(* IEC 61131-3 sources: volt/packages/volt-lsp-iec/test-corpus/lenze-mid/Device/Plc Logic/Application/Library Manager/L_FirstErrorCapture, 3.26.2.8 (Lenze), 36 files *)

(* ---- ENUMSTEPSFILEHANDLING.dut ---- *)
TYPE ENUMSTEPSFILEHANDLING :
(
	INIT := 0,
	OPENFILE := 1,
	GETSIZEFILE := 2,
	READFILE := 3,
	WAITREAD := 4,
	WAITCLOSE := 5,
	CLOSEFILE := 6,
	DONE := 7
);
END_TYPE

(* ---- SCCATEGORYSTRUCT.dut ---- *)
TYPE SCCATEGORYSTRUCT :
STRUCT
	ASSTR : ARRAY [0..uiNoOfDowntimeCategories] OF STRING(55);
	AXERROR : ARRAY [0..uiNoOfDowntimeCategories] OF BOOL;
END_STRUCT
END_TYPE

(* ---- SCERRORACCESS.dut ---- *)
TYPE SCERRORACCESS :
STRUCT
	DWCATEGORY : DWORD;
	WERRORCODE : WORD;
	ETYPE : INT;
	STEXT : STRING;
END_STRUCT
END_TYPE

(* ---- SCERRORDATA.dut ---- *)
TYPE SCERRORDATA :
STRUCT
	XFIRSTERRORACTIVE : BOOL;
	XISWARNINGINFO : BOOL;
	IPRIORITY : INT;
	DWERRORNUMBER : DWORD;
END_STRUCT
END_TYPE

(* ---- SCERRORDATA_BASE.dut ---- *)
TYPE SCERRORDATA_BASE :
STRUCT
	SERRDESC : STRING;
	SCATEGORYDESC : STRING(55);
	DWERRORCATEGORY : DWORD;
	IPRODUCTIONEVENTMODE : INT;
	XCATEGORYERROR : BOOL;
END_STRUCT
END_TYPE

(* ---- SCREADERRORFROMFILEIN.dut ---- *)
TYPE SCREADERRORFROMFILEIN :
STRUCT
	SFILENAME : FILE.CAA.FILENAME := 'SoftPlcParameter/SoftPlcParameter.lxd';
	IMAXREADLOOPS : INT := 1;
	WTEXTLISTID : WORD := 15360;
	WENDTEXTLISTID : WORD := 16383;
	WERRORID : WORD := 1;
END_STRUCT
END_TYPE

(* ---- SCREADERRORFROMFILEOUT.dut ---- *)
TYPE SCREADERRORFROMFILEOUT :
STRUCT
	WFINDTEXTLISTID : WORD;
	WFINDERRORID : WORD;
	DIREADROWS : DINT;
	DIERRORROWS : DINT;
	SERRORTEXT : STRING(255);
	XEOF : BOOL;
	TEXCUTETIME : TIME;
	STEP : enumStepsFileHandling;
	STATUS : scRearErrorfromFileStatus;
END_STRUCT
END_TYPE

(* ---- SCREARERRORFROMFILESTATUS.dut ---- *)
TYPE SCREARERRORFROMFILESTATUS :
STRUCT
	XDONEOPENFILE : BOOL;
	XBUSYOPENFILE : BOOL;
	XERROROPENFILE : BOOL;
	EOPENFILEERROR : FILE.ERROR;
	HFILE : FILE.CAA.HANDLE;
	XDONEGETSIZEFILE : BOOL;
	XBUSYGETSIZEFILE : BOOL;
	XERRORGETSIZEFILE : BOOL;
	EGETSIZEFILEERROR : FILE.ERROR;
	SZSIZE : FILE.CAA.SIZE;
	XDONEREADFILE : BOOL;
	XBUSYREADFILE : BOOL;
	XERRORREADFILE : BOOL;
	EREADFILEERROR : FILE.ERROR;
	XDONECLOSEFILE : BOOL;
	XBUSYCLOSEFILE : BOOL;
	XERRORCLOSEFILE : BOOL;
	ECLOSEFILEERROR : FILE.ERROR;
	XDONEFINDERROR : BOOL;
	XBUSYFINDERROR : BOOL;
	XERRORFINDERROR : BOOL;
END_STRUCT
END_TYPE

(* ---- SCTM_FB_ERROR.dut ---- *)
TYPE SCTM_FB_ERROR :
STRUCT
	XAXISERROR : BIT;
	XAXISWARNING : BIT;
	XDRIVEERROR : BIT;
	XDRIVEWARNING : BIT;
	IERRORID : INT;
	DWDRIVEERROR : DWORD;
END_STRUCT
END_TYPE

(* ---- UERRORNUMBER.dut ---- *)
TYPE UERRORNUMBER :
UNION
	DWERRORNUMBER : DWORD;
	AWERRORINFO : ARRAY [1..2] OF WORD;
END_UNION
END_TYPE

(* ---- GVL_ERRCAPT.gvl ---- *)
VAR_GLOBAL
	IUDINTQTY : INT := 4;
	IERRORQTY : INT := 160;
	IERRCATEGORY : INT := 99;
END_VAR

(* ---- GVL_FIRSTERRORLOCAL.gvl ---- *)
VAR_GLOBAL
	UINOOFDOWNTIMECATEGORIES : UINT := 99;
END_VAR

(* ---- GVL_READERRORFROMFILE.gvl ---- *)
VAR_GLOBAL
	IMAXERRORTEXTARRAYSIZE : INT := 1250;
	IMAXREADSIZE : INT := 80;
	ASERRORTEXT : ARRAY [0..GVL_ReadErrorFromFile.imaxErrorTextArraySize] OF STRING(255);
	ADWERRORID : ARRAY [0..GVL_ReadErrorFromFile.imaxErrorTextArraySize] OF DWORD;
END_VAR

(* ---- GETAPPLICATIONTERRORSTRING.pou ---- *)
FUNCTION GETAPPLICATIONTERRORSTRING : STRING(255)
VAR_INPUT
	WTEXTREFID : WORD;
	WERRORID : WORD;
	DWERRORNUMBER : DWORD;
END_VAR
END_FUNCTION

(* ---- GETDATETIMEFROMJSON.pou ---- *)
FUNCTION GETDATETIMEFROMJSON : STRING
VAR_INPUT
	XUSEMILLISECONDS : BOOL;
END_VAR
VAR_IN_OUT
	SJSONSTRING : STRING(255);
END_VAR
END_FUNCTION

(* ---- GETDRIVEERRORSTRING.pou ---- *)
FUNCTION GETDRIVEERRORSTRING : STRING(255)
VAR_INPUT
	WTEXTREFID : WORD;
	WERRORID : WORD;
	DWERRORNUMBER : DWORD;
END_VAR
END_FUNCTION

(* ---- GETDWREASONCODEFROMJSON.pou ---- *)
FUNCTION GETDWREASONCODEFROMJSON : DWORD
VAR_IN_OUT
	SJSONSTRING : STRING(255);
END_VAR
END_FUNCTION

(* ---- GETFASTERRORSTRING.pou ---- *)
FUNCTION GETFASTERRORSTRING : STRING(255)
VAR_INPUT
	WTEXTREFID : WORD;
	WERRORID : WORD;
	DWERRORNUMBER : DWORD;
END_VAR
END_FUNCTION

(* ---- GETREASONCODESTRINGFROMJSON.pou ---- *)
FUNCTION GETREASONCODESTRINGFROMJSON : STRING
VAR_IN_OUT
	SJSONSTRING : STRING(255);
END_VAR
END_FUNCTION

(* ---- SEVERITYTOPRIORITY.pou ---- *)
FUNCTION SEVERITYTOPRIORITY : INT
VAR_INPUT
	ESEVERITY : L_IE1P_SeverityLevel;
END_VAR
END_FUNCTION

(* ---- L_ERRCAPTUDINT.pou ---- *)
FUNCTION_BLOCK L_ERRCAPTUDINT
VAR_INPUT
	UDIERROR : UDINT;
	ASCERRORDATA : ARRAY [0..31] OF scErrorData;
	XRESET : BOOL;
END_VAR
VAR_OUTPUT
	XERRORACTIVE : BOOL;
	SCFIRSTERROR : scErrorData;
END_VAR
VAR
	AXERROR : ARRAY [0..31] OF BOOL;
	AIINDEX : ARRAY [1..4] OF INT;
	XITERATIONDONE : BOOL;
END_VAR
END_FUNCTION_BLOCK

(* ---- L_FINDERRORINFILE.pou ---- *)
FUNCTION_BLOCK L_FINDERRORINFILE
VAR_INPUT
	ISIZE : INT;
	XEXECUTE : BOOL;
	WTEXTLISTID : WORD;
	WENDTEXTLISTID : WORD;
	WERRORID : WORD;
	XSTOREALLERRORTEXT : BOOL;
	XTEXREFIDERRORONLY : BOOL;
	XSTOREALLAPPTEXREFIDERRORTEXT : BOOL;
	XSTOPIFERRORFOUND : BOOL;
END_VAR
VAR_OUTPUT
	SERRORLINE : STRING(255);
	SERRORTEXT : STRING(255);
	DIREADROW : DINT;
	DIERRORROW : DINT;
	XFINDERROR : BOOL;
	XDONE : BOOL;
	XBUSY : BOOL;
	XERROR : BOOL;
	WFINDTEXTLISTID : WORD;
	WFINDERRORID : WORD;
	STEXTLISTID : STRING;
	SERRORID : STRING;
END_VAR
VAR_IN_OUT
	AREADBUFFERARRAY : ARRAY [0..GVL_ReadErrorFromFile.imaxReadSize] OF BYTE;
	ASERRORTEXT : ARRAY [0..GVL_ReadErrorFromFile.imaxErrorTextArraySize] OF STRING(255);
	ADWERRORID : ARRAY [0..GVL_ReadErrorFromFile.imaxErrorTextArraySize] OF DWORD;
END_VAR
VAR
	SREADFROMFILE : STRING(255);
	SREADLINE : STRING(255);
	CHARXX : STRING(1);
	I : INT;
	XMEMMOVERECEIVE : BOOL;
	ICRLFPOS : INT;
	RT_EXECUTE : R_TRIG;
END_VAR
END_FUNCTION_BLOCK

METHOD METHEXTRACTERROR : BOOL
VAR_INPUT
	TEXREFIDERRORONLY : BOOL;
	XSTOREALLAPPTEXREFIDERRORTEXT : BOOL;
END_VAR
VAR_IN_OUT
	SERRORLINE : STRING(255);
	SERRORTEXT : STRING(255);
	WTEXTLISTID : WORD;
	WENDTEXTLISTID : WORD;
	WERRORID : WORD;
	WFINDTEXTLISTID : WORD;
	WFINDERRORID : WORD;
	STEXTLISTID : STRING;
	SERRORID : STRING;
	DIERRORROW : DINT;
END_VAR
END_METHOD

(* ---- L_FIRSTERRCAPTURE.pou ---- *)
FUNCTION_BLOCK L_FIRSTERRCAPTURE
VAR_INPUT
	XRESETFIRSTERRCAPTURE : BOOL;
END_VAR
VAR_OUTPUT
	XERRORACTIVE : BOOL;
	SCFIRSTERRORDATA : scErrorData;
END_VAR
VAR_IN_OUT
	AUDIERRORBITS : ARRAY [0..GVL_ErrCapt.iUDINTQty] OF UDINT;
	ASCERRORDATA : ARRAY [0..GVL_ErrCapt.iErrorQty] OF scErrorData;
END_VAR
VAR
	MASTERERRCAPT : L_ErrCaptUDINT;
	AERRCAPTUDINT : ARRAY [0..GVL_ErrCapt.iUDINTQty] OF L_ErrCaptUDINT;
	AIINDEX : ARRAY [1..4] OF INT;
	TONRESETTIMER : TON;
	RTRIGRESET : R_TRIG;
END_VAR
END_FUNCTION_BLOCK

(* ---- L_FIRSTERRCAPTUREERRORACCESS.pou ---- *)
FUNCTION_BLOCK L_FIRSTERRCAPTUREERRORACCESS
VAR_INPUT
	XENABLE : BOOL;
	XPRIOFROMERROR : BOOL;
	XRESETFIRSTERRCAPTURE : BOOL;
	SCERRORACCESS : scErrorAccess;
	IPRODUCTIONMODE : INT;
END_VAR
VAR_OUTPUT
	XBUSY : BOOL;
	XERRORACTIVE : BOOL;
	XUPDATEERROR : BOOL;
	XISWARNINGINFO : BOOL;
	SCFIRSTERRORDATA : scErrorData;
	XERRORFB : BOOL;
END_VAR
VAR_IN_OUT
	ACATEGORYSTRING : scCategoryStruct;
END_VAR
VAR
	DWLASTCATEGORY : DWORD;
	DWLASTERRORNUMBER : DWORD;
	TRIGUPDATE : F_TRIG;
END_VAR
END_FUNCTION_BLOCK

(* ---- L_FIRSTERRCAPTURESETERRORSINGLE.pou ---- *)
FUNCTION_BLOCK L_FIRSTERRCAPTURESETERRORSINGLE
VAR_INPUT
	XRESETFIRSTERRCAPTURE : BOOL;
	UIMAXERROR : UINT;
END_VAR
VAR_OUTPUT
	XERRORACTIVE : BOOL;
	SCFIRSTERRORDATA : scErrorData;
END_VAR
VAR_IN_OUT
	ASCERRORINFO : ARRAY [0..GVL_ErrCapt.iErrorQty] OF L_IE1P_ErrorInfo;
	ASCADDERRORINFO : ARRAY [0..GVL_ErrCapt.iErrorQty] OF scErrorData_base;
END_VAR
VAR
	FBFIRSTERRSETERRORSINGLE : L_FirstErrCapture;
	AUERRORNUMBER : ARRAY [0..GVL_ErrCapt.iErrorQty] OF uErrorNumber;
	ASCERRORDATA : ARRAY [0..GVL_ErrCapt.iErrorQty] OF scErrorData;
	AUDIERRORBITS : ARRAY [0..GVL_ErrCapt.iUDINTQty] OF UDINT;
	AUDIERRORBITSRESET : ARRAY [0..GVL_ErrCapt.iUDINTQty] OF UDINT;
	IINDEX : INT;
	XFCERROR : BOOL;
	IMAXERRORLOOP : INT;
	XERRORBIT : BOOL;
END_VAR
END_FUNCTION_BLOCK

METHOD CONV_INDEX_TO_BITX : BOOL
VAR_INPUT
	XERRORBIT : BOOL;
	IINDEX : INT;
END_VAR
END_METHOD

(* ---- L_FIRSTFASTERRCAPTURE.pou ---- *)
FUNCTION_BLOCK L_FIRSTFASTERRCAPTURE
VAR_INPUT
	XENABLE : BOOL;
	SCFASTERRORINFO : L_IE1P_ErrorInfo;
	SCFASTADDERRORINFO : scErrorData_base;
	XACTIVATEFASTERRORINPUT : BOOL := TRUE;
	XCAPTUREALLREASON : BOOL := TRUE;
	XCAPTUREONLYFASTERROR : BOOL := TRUE;
	XCAPTURESTOREWARNING_LOCK : BOOL := FALSE;
	XPRIOFROMERROR : BOOL := TRUE;
	XRESETFIRSTERRCAPTURE : BOOL;
	UIMAXERROR : UINT;
	IPRODUCTIONMODE : INT;
END_VAR
VAR_OUTPUT
	XBUSY : BOOL;
	XERRORACTIVE : BOOL;
	XFASTERRORACTIVE : BOOL;
	XUPDATEERROR : BOOL;
	XISWARNINGINFO : BOOL;
	SCFIRSTERRORDATA : scErrorData;
END_VAR
VAR_IN_OUT
	ASCERRORINFO : ARRAY [0..GVL_ErrCapt.iErrorQty] OF L_IE1P_ErrorInfo;
	ASCADDERRORINFO : ARRAY [0..GVL_ErrCapt.iErrorQty] OF scErrorData_base;
END_VAR
VAR
	SCERRORDATARESET : scErrorData;
	IHIGHESTPRIO : INT;
	IINDEX : INT;
	IINDEXHIGHESTPRIO : INT;
	IMAXERRORLOOP : INT;
	XERRORSET : BOOL;
	TRIGUPDATE : F_TRIG;
	IWARNING_LOCK : INT := 7;
	IWARNING : INT := 8;
	IWARNINGINFO : INT;
	XWARNINGINFOGONE : BOOL;
	ILASTHIGHPRIORITY : INT;
	ILASTINDEXHIGHESTPRIO : INT;
END_VAR
END_FUNCTION_BLOCK

(* ---- L_GETERRORTEXTFROMFILEREADARRAY.pou ---- *)
FUNCTION_BLOCK L_GETERRORTEXTFROMFILEREADARRAY
VAR_INPUT
	XENABLED : BOOL;
	XERRORACTIVE : BOOL;
	XUPDATEERROR : BOOL;
	XONLYUSERAPPERRORFROMFILE : BOOL;
	SCFIRSTERRORDATA : scErrorData;
	IMAXNOOFSEARCHLOOPS : INT;
END_VAR
VAR_OUTPUT
	SCFIRSTERRORDATAOUT : scErrorData;
	DWFINDERRORID : DWORD;
	IERRORINDEX : INT;
	SERRORTEXT : STRING(255);
	ISEARCHLOOPS : INT;
	XERRORTEXTFROMFUN : BOOL;
END_VAR
VAR_IN_OUT
	ASERRORTEXT : ARRAY [0..GVL_ReadErrorFromFile.imaxErrorTextArraySize] OF STRING(255);
	ADWERRORID : ARRAY [0..GVL_ReadErrorFromFile.imaxErrorTextArraySize] OF DWORD;
END_VAR
VAR
	RTRIG_XERRORACTIVE : R_TRIG;
	ISEARCHINDEX : INT;
	ICMPINDEX : INT;
	INOOFSEARCHLOOPS : INT;
	WTEXTREFID : WORD;
	WERRORID : WORD;
END_VAR
END_FUNCTION_BLOCK

(* ---- L_GETERRORTEXTFROMFUNCTION.pou ---- *)
FUNCTION_BLOCK L_GETERRORTEXTFROMFUNCTION
VAR_INPUT
	XENABLED : BOOL;
	XERRORACTIVE : BOOL;
	XUPDATEERROR : BOOL;
	SCFIRSTERRORDATA : scErrorData;
END_VAR
VAR_OUTPUT
	SCFIRSTERRORDATAOUT : scErrorData;
	SERRORTEXT : STRING(255);
	XERRORTEXTFROMFUN : BOOL;
END_VAR
VAR
	RTRIG_XERRORACTIVE : R_TRIG;
	WTEXTREFID : WORD;
	WERRORID : WORD;
END_VAR
END_FUNCTION_BLOCK

(* ---- L_GETERRORTEXTFROMHMI.pou ---- *)
FUNCTION_BLOCK L_GETERRORTEXTFROMHMI
VAR_INPUT
	XENABLED : BOOL;
	XERRORACTIVE : BOOL;
	XUPDATEERROR : BOOL;
	SCFIRSTERRORDATA : scErrorData;
	TMAXWAITTIME : TIME := TIME#5s0ms;
	SACTUALPLCREASONCODE : STRING(255);
END_VAR
VAR_OUTPUT
	XBUSY : BOOL;
	XDONE : BOOL;
	XERRORACTIVEDELAYED : BOOL;
	SCFIRSTERRORDATAOUT : scErrorData;
	XFINDERRORID : BOOL;
	TTIMEFIND : TIME;
	SERRORTEXT : STRING(255);
END_VAR
VAR_IN_OUT
	SACTUALVISUREASONCODE : STRING(255);
END_VAR
VAR
	RTRIG_XERRORACTIVE : R_TRIG;
	TERRORACTIVETIME : TON;
	SCUTSTRING : STRING(255);
	DTPLCDATETIME : DATE_AND_TIME;
	DTHMIDATETIME : DATE_AND_TIME;
	DTLASTPLCDATETIME : DATE_AND_TIME;
	SPLCDATETIME : STRING;
	SHMIDATETIME : STRING;
	XONEWAITINGPLCCYCLE : BOOL;
	DWPLCREASONCODE : DWORD;
	SERRORTEXTMONITOR : STRING(255);
END_VAR
END_FUNCTION_BLOCK

(* ---- L_OVERWRITEFIRSTERRCAPTURE.pou ---- *)
FUNCTION_BLOCK L_OVERWRITEFIRSTERRCAPTURE
VAR_INPUT
	XENABLE : BOOL;
	SCFIRSTERRORDATA : scErrorData;
	SCERRORINFO : L_IE1P_ErrorInfo;
	SCADDERRORINFO : scErrorData_base;
	IPRODUCTIONMODE : INT;
END_VAR
VAR_OUTPUT
	XERROROVERWRITEACTIVE : BOOL;
	XERRORACTIVE : BOOL;
	XUPDATEERROR : BOOL;
	XISWARNINGINFO : BOOL;
	SCOUTFIRSTERRORDATA : scErrorData;
END_VAR
VAR
	SCTEMPFIRSTERRORDATA : scErrorData;
	R_TRIGUPDATEXENABLE : R_TRIG;
	R_TRIGUPDATEXERROR : R_TRIG;
	F_TRIGUPDATEXENABLE : F_TRIG;
	F_TRIGUPDATEXERROR : F_TRIG;
END_VAR
END_FUNCTION_BLOCK

(* ---- L_READERRORFROMFILE.pou ---- *)
FUNCTION_BLOCK L_READERRORFROMFILE
VAR_INPUT
	XENABLE : BOOL;
	XEXECUTE : BOOL;
	XSTOREALLERRORTEXT : BOOL;
	XSTORETEXREFIDERRORTEXT : BOOL;
	XSTOREALLAPPTEXREFIDERRORTEXT : BOOL;
	XSTOPIFERRORFOUND : BOOL;
	XCONTINUOUSREAD : BOOL;
	XREPEAT : BOOL;
	XINIT : BOOL;
	XCLEARERRORARRAYS : BOOL;
	SCIN : scReadErrorFromFileIN;
END_VAR
VAR_OUTPUT
	XFINDERROR : BOOL;
	XERROR : BOOL;
	XBUSY : BOOL;
	XDONE : BOOL;
	SCOUT : scReadErrorfromFileOUT;
END_VAR
VAR_IN_OUT
	ASERRORTEXT : ARRAY [0..GVL_ReadErrorFromFile.imaxErrorTextArraySize] OF STRING(255);
	ADWERRORID : ARRAY [0..GVL_ReadErrorFromFile.imaxErrorTextArraySize] OF DWORD;
END_VAR
VAR
	OPENFILE : FILE.Open;
	XEXEOPENFILE : BOOL;
	EFILEMODE : FILE.MODE;
	GETSIZEFILE : FILE.GetSize;
	XEXEGETSIZEFILE : BOOL;
	READFILE : FILE.Read;
	XEXEREADFILE : BOOL;
	XABORTREADFILE : BOOL;
	UDITIMEOUTREADFILE : UDINT;
	XABORTEDREADFILE : BOOL;
	PBUFFERREADFILE : FILE.CAA.PVOID;
	SZBUFFERREADFILE : FILE.CAA.SIZE;
	SZSIZEREADFILE : FILE.CAA.SIZE;
	AREADBUFFERARRAY : ARRAY [0..GVL_ReadErrorFromFile.imaxReadSize] OF BYTE;
	CLOSEFILE : FILE.Close;
	XEXECLOSEFILE : BOOL;
	FBFINDERRORINFILE : L_FindErrorInFile;
	XEXEFINDERROR : BOOL;
	SERRORLINE : STRING(255);
	XSTARTWAITTIME : BOOL;
	XSTARTREADTIME : BOOL;
	TONWAITTIME : TON;
	TONREADTIME : TON;
	XFIRSTINIT : BOOL;
	TONEXECUTETIME : TON;
	XSTARTEXECUTETIMER : BOOL;
	I : INT;
	RTRIGXEXECUTE : R_TRIG;
END_VAR
END_FUNCTION_BLOCK

(* ---- L_SETERRORSINGLE_TM_FB.pou ---- *)
FUNCTION_BLOCK L_SETERRORSINGLE_TM_FB
VAR_INPUT
	XCAPTUREONLYFASTERROR : BOOL := TRUE;
	SCTM_FB_ERROR : scTM_FB_Error;
	DWERRORCATEGORY : DWORD;
END_VAR
VAR_OUTPUT
	SCERRORINFO : L_IE1P_ErrorInfo;
	SCADDERRORINFO : scErrorData_base;
END_VAR
VAR_IN_OUT
	ASERRORCATEGORY : ARRAY [0..GVL_ErrCapt.iErrCategory] OF STRING(55);
	AXERRORCATEGORY : ARRAY [0..GVL_ErrCapt.iErrCategory] OF BOOL;
END_VAR
VAR
	DWERRORCATEGORYCHECK : DWORD;
END_VAR
END_FUNCTION_BLOCK

(* ---- L_SETERRORSINGLEADDINFO.pou ---- *)
FUNCTION_BLOCK L_SETERRORSINGLEADDINFO
VAR_INPUT
	DWERRORCATEGORY : DWORD;
END_VAR
VAR_OUTPUT
	ASCADDERRORINFO : scErrorData_base;
END_VAR
VAR_IN_OUT
	ASERRORCATEGORY : ARRAY [0..GVL_ErrCapt.iErrCategory] OF STRING(55);
	AXERRORCATEGORY : ARRAY [0..GVL_ErrCapt.iErrCategory] OF BOOL;
END_VAR
VAR
	DWERRORCATEGORYCHECK : DWORD;
END_VAR
END_FUNCTION_BLOCK

(* ---- L_SETERRORSINGLEINFO.pou ---- *)
FUNCTION_BLOCK L_SETERRORSINGLEINFO
VAR_INPUT
	SERRORDESCRIPTION : STRING(55);
	DWERRORCATEGORY : DWORD;
END_VAR
VAR_OUTPUT
	ASCADDERRORINFO : scErrorData_base;
END_VAR
VAR_IN_OUT
	ASERRORCATEGORY : ARRAY [0..GVL_ErrCapt.iErrCategory] OF STRING(55);
END_VAR
VAR
	DWERRORCATEGORYCHECK : DWORD;
END_VAR
END_FUNCTION_BLOCK

(* ---- L_SETFASTERRORSINGLEADDINFO.pou ---- *)
FUNCTION_BLOCK L_SETFASTERRORSINGLEADDINFO
VAR_INPUT
	XMODULCATEGORYDESC : BOOL;
	SERRORCATEGORY : STRING(55);
	DWERRORCATEGORY : DWORD;
END_VAR
VAR_OUTPUT
	ASCERRORINFO : L_IE1P_ErrorInfo;
	SCADDERRORINFO : scErrorData_base;
END_VAR
VAR_IN_OUT
	ASERRORCATEGORY : ARRAY [0..GVL_ErrCapt.iErrCategory] OF STRING(55);
	AXERRORCATEGORY : ARRAY [0..GVL_ErrCapt.iErrCategory] OF BOOL;
END_VAR
VAR
	DWERRORCATEGORYCHECK : DWORD;
END_VAR
END_FUNCTION_BLOCK

(* ---- L_SETFASTERRORSINGLEINFO.pou ---- *)
FUNCTION_BLOCK L_SETFASTERRORSINGLEINFO
VAR_INPUT
	XERRORACTIVE : BOOL;
	DWERRORCODE : DWORD;
	ESEVERITY : L_IE1P_SeverityLevel;
END_VAR
VAR_OUTPUT
	SCERRORINFO : L_IE1P_ErrorInfo;
END_VAR
END_FUNCTION_BLOCK
